{attribute 'analysis' := '-33'}
PROGRAM PRG_HelperTests
VAR
{IF defined (UNIT_TEST)}
    fbF_ToAnyBytesTests        : FB_F_ToAnyBytesTests;
{END_IF}
END_VAR

END_PROGRAM

(* stored: Version 1.1.0.1
   POU PRG_HelperTests: Id {1b1594ec-42ab-49ac-9789-def7d70c2333}, SpecialFunc None *)
